// TIA Portal V16 export
// export: Created 2026-06-17T17:21:10.394091Z, ExportSetting WithDefaults, DisplayName Totally Integrated Automation Portal, DisplayVersion V16 Update 8, DisplayName TIA Portal Version Control Interface, DisplayVersion V16 Update 8, DisplayName TIA Portal Openness, DisplayVersion V16 Update 8, DisplayName SINAMICS Startdrive Advanced, DisplayVersion V16, DisplayName SINAMICS Startdrive G130, G150, S120, S150, SINAMICS MV, S210, DisplayVersion V16, DisplayName SINAMICS Startdrive G110M, G120, G120C, G120D, G120P, DisplayVersion V16, DisplayName STEP 7 Professional, DisplayVersion V16 Update 8, DisplayName STEP 7 Safety, DisplayVersion V16 Update 7, DisplayName WinCC Advanced, DisplayVersion V16 Update 8
Screen "Temperature_Monitor"  1280x800, Number=1
  ScreenLayer 
    IOField "IO_Temp3" at 240,460 size 140x44  DataFormat=Decimal, FormatPattern=9999999, Mode=InOutput
    Button "BTN_Reset3" at 540,460 size 100x44  Mode=Text, HelpText="复位", TextOff="Text", TextOn="Text"
    SymbolicIOField "SIO_Status" at 930,140 size 160x44  CountVisibleItems=3, Mode=InOutput, OnValue=1, TextOff="0", TextOn="1"
    Circle "LMP_OH3" at 430,468 size 48x48
    TextField "TXT_Status" at 800,140 size 120x40  Text="系统状态Text"
